Staubli VAL3: IsInTheSameBox.pgx

program IsInTheSameBox(bool& x_bFindInBox1[], string& x_sLodaBox1[], bool& x_bInBox1[])
  local num i
  local num l_nNum
begin
  l_nNum=1
  resize(nInWhichBox,1,1)
  nInWhichBox=-1
  for i=0 to size(x_bFindInBox1)-1
    if x_bFindInBox1[i]==true
      x_bInBox1=true
      if nInWhichBox[size(nInWhichBox)-1]==-1
        nInWhichBox=i
      else
        $dins(nInWhichBox,size(nInWhichBox))
        nInWhichBox[size(nInWhichBox)-1]=i
      endIf
    endIf
  endFor
  if size(nInWhichBox)==1
    x_sLodaBox1=sBox1[nInWhichBox]
  else
    call findInWhichBox1(x_sLodaBox1)
  endIf

end
